Universal Robots URScript: SUB_3100.script

def SUB_3100():
  global _hidden_verificationVariable=0
  set_standard_analog_input_domain(0, 1)
  set_standard_analog_input_domain(1, 1)
  set_tool_analog_input_domain(0, 1)
  set_tool_analog_input_domain(1, 1)
  set_analog_outputdomain(0, 0)
  set_analog_outputdomain(1, 0)
  set_input_actions_to_default()
  set_runstate_gp_boolean_output_to_value(0, 3)
  set_safety_mode_transition_hardness(1)
  set_tcp(p[0.0,0.06,0.535,0.0,0.0,0.0])
  set_gravity([0.0, 0.0, 9.82])
  set_tool_communication(False, 115200, 0, 1, 1.5, 3.5)
  set_tool_output_mode(0)
  set_tool_digital_output_mode(0, 1)
  set_tool_digital_output_mode(1, 1)
  set_tool_voltage(0)
  set_target_payload(0.100000, [0.135000, 0.000000, 0.225000], [10.000000, 10.000000, 10.000000, 0.000000, 0.000000, 0.000000])
  global isReCapt=False
  global Bucket_Z=[0, 0.7]
  global DistPillar=475
  global CandCnt=0
  global lr=1
  global ReCaptZ=0.05
  global forceval=p[0, 0, 0, 0, 0, 0]
  global CaptDepth=[0.24, 0.72, 0]
  global port=3000
  global isOnlyF=True
  global retX2=p[-0.09927, 0.42868, -0.30877, 0.00019, -0.00018, -1.59231]
  global socket_timeout=120
  global isSkipP=False
  global curpos=p[0, 0, 0, 0, 0, 0]
  global host="192.168.1.2"
  global is_popup=False
  global CaptZOffset=0
  global isGoHome=True
  global i_pos2=p[-0.73669, 0.09787, -0.42767, 2.01816, 2.03864, 0.34287]
  global i_pos1=p[-0.73588, 0.09792, -0.42776, 2.01775, 2.03812, 0.34393]
  global pBucket=[p[0.82431, 0.40374, 0.29254, 0, 0, -1.56059], p[-0.84041, -0.48526, 0.27877, 0, 0, 1.6028], p[0, 0, 0, 0, 0, 0]]
  global CaptStepZ=0.08
  global CaptIndex=[0, 0, 0]
  global CaptStepX=0.432
  global pBucketM=p[-0.80141, -0.42542, 0.2879, 0, 0, 1.55713]
  global socket_name="vt"
  global rovi_err=0
  global SubPrgResult=820
  global CurrPos=p[-0.89356, -0.02064, 0.55405, 2.21465, 2.1843, 0.05997]
  global CurrPos_p=p[-0.80753, -0.01858, 0.02262, 2.21465, 2.1843, 0.05997]
  global ForceStartZ=0.43553
  global CutOffZ=0.08
  global HomeDistTh=0.05
  global RBDistTh=0.05
  global RBRadiusTh=0.3
  global RBXTh=[-0.5, 0.5]
  global RBYTh=[-0.8, 1]
  global RBZTh=[-0.1, 0.1]
  global Sub3100_ZMax=0.74
  global ForceStartX=-0.98868
  global Sub3100_aRot=0.2
  global Sub3100_d=0.3
  global Sub3100_Option=18
  global Sub3100_a=0.2
  global Sub3100_XdV=0.1
  global Sub3100_XdRot=8
  global ZoneDistTh=0.05
  global ZoneRadiusTh=0.3
  global ZoneXTh=[-0.5, 0.5]
  global ZoneYTh=[-0.8, 1]
  global ZoneZTh=[-0.1, 0.1]
  global BucketWidth=0.95
  global ZoneBucketGap=0.1
  global ZoneHomeX=[-0.2, 0.2]
  global UnloadZ=0.05
  global CaptPos=p[-0.42193,-0.00317,0.36000,2.199,2.246,0.022]
  global BucketUpperPos=p[0.42193,0.00317,0.36000,2.199,2.246,0.022]
  global Sub3100_GPII18=0
  global Bucket=p[0.32604,0.49174,0.0,-1.882900624652718E-5,2.8304179127934987E-5,-1.593185305749222]
  global BucketM=p[0.32604,0.49174,0.0,1.2814539732933814E-16,-2.611297964559462E-16,-1.5931853071795858]
  global CaptPoint_C=p[-0.4219337985373468,-0.003168602281063755,0.36,-2.1962364319979395,-2.2439316084554193,-0.02184884826814999]
  global CaptPoint_C2=p[0.32796661698047924,-0.010768520544682924,0.01931625281283378,2.2288103429550152,-2.213636886217198,8.598462540813273E-5]
  global CaptPoint_L1=p[-0.42193494849366175,-0.2,0.36,-2.1962086037526616,-2.243896582262281,-0.02199725151102503]
  global CaptPoint_L2=p[0.327894307417917,-0.010799940826224014,0.01928712668893995,2.087717047309385,-2.0736781215133306,0.27365839887453103]
  global CaptPoint_R1=p[-0.4219551896101372,0.3,0.36,-2.1960823751566156,-2.243954123514977,-0.021863042557794844]
  global CaptPoint_R2=p[0.327926308680866,-0.010795166414457658,0.019300245403843563,-2.1186306375223185,2.1040550557443427,0.22023197678473694]
  global Capt_1BK_L=p[-0.4574214308482636,-0.48457071473611046,0.3504487959434708,-2.1962343446504526,-2.243967222238911,-0.021809195357489434]
  global Capt_1BK_L_kari=p[-0.9062780457975316,-0.3948152887685301,0.3041579389647211,-1.973454285761923,-1.9354309814821136,0.46582663599327684]
  global Capt_1BK_R=p[-0.4574597285646511,0.4755214243904677,0.35039311859649847,-2.196330286580149,-2.2438949166739053,-0.021738621025254933]
  global Capt_1BK_R_kari=p[-0.9062432457725078,0.5951337546911526,0.30410336812750105,-1.9735777661712788,-1.9353884348839347,0.46584435471052615]
  global Capt_1BK_pos1=p[-0.4218793038724447,-0.003154429464978058,0.2915499891144615,-2.1963422029204875,-2.2438663520270015,-0.02197160668673838]
  global Capt_1BK_pos2=p[-0.42187829024618434,-0.0031710253373066375,0.29156503858953065,-2.196324918349679,-2.2439040699490773,-0.021928444416953782]
  global Capt_1BK_pos2_k=p[-0.6125678682784722,-0.030388805985305904,0.07817890571333086,-1.7892541925095446,-1.8765982468297469,0.6168577595976025]
  global Capt_2BK_L=p[0.42186661528427194,0.4254738068040517,0.35042275762909847,2.239156309475874,-2.1837044610999294,0.002643817066643282]
  global Capt_2BK_L_kari=p[1.0654977997166857,0.48819520122022786,0.0997150581225536,-1.8581624430714432,1.7479280549699192,-0.330138866280949]
  global Capt_2BK_R=p[0.4218208572756906,-0.5427676723257963,0.350372239919558,2.2392697861179327,-2.183553596194912,0.002410470905346486]
  global Capt_2BK_R_kari=p[1.0635189639466671,-0.5406292885234477,0.09156512141204048,-2.1417082668537115,1.7859902718169367,-0.7309097134650204]
  global Capt_2BK_pos1=p[0.42193501458435656,0.004742683868356356,0.35045865974037793,2.2391012408536453,-2.1839704655717003,0.002677867056024068]
  global Capt_2BK_pos2=p[0.421903984494575,0.004707988774967922,0.35045218900915065,2.239114367170047,-2.183895515396197,0.002684056681074047]
  global Capt_2BK_pos2_k=p[0.4977433025854323,-0.009744988529796803,0.07805101846052531,-1.951106747250682,1.9044153054141988,-0.5362260997480872]
  global Capt_GD_M=p[-0.004067001529315755,-0.25244814937804905,-2.093072695775744E-4,0.0332905748643788,-3.1401478399413327,-0.0037841799742876323]
  global Depart_1GD=p[2.9272629556870893E-4,-0.32809839693864495,0.01933497371622539,0.06378642771012696,-3.140731101950783,-3.370184732371461E-4]
  global Depart_LM_2GD=p[-0.022329487227551487,-0.6428077701737687,0.030336146545121845,-0.0656618547018821,2.9888986438241005,0.1566836156643787]
  global Depart_M=p[0.03703236558231149,-0.6428132409158767,-0.02112384231382136,-0.05669816428100925,3.1320592135794345,0.16829522075932857]
  global Depart_RM_2GD=p[0.10304778501057178,-0.6389514408512296,0.030085893950939302,0.039485966396909634,-3.0126453050861945,-0.17126767917269797]
  global Depsrt_2GD=p[3.027477292580124E-4,-0.3281073069657892,0.019292078494201337,0.06380062875024692,-3.1406974312388685,-3.876005598966342E-4]
  global HomePointL=p[-0.36789,-0.5117344641471838,0.78,-0.6278857271586024,3.0680899128661667,-8.649957362498864E-4]
  global PickPos=p[0.10830682331105715,-1.3709505888096256,-0.18404188875951455,-0.00622194000158997,2.880236948927292,-0.00383636509397631]
  global Solve=p[-0.00368,-0.0021000000000000003,0.25739999999999996,0.0,0.0,0.0]
  global TEST=p[0.1,0.0,0.2,0.0,0.0,0.0]
  global UF=p[0.0,0.0,0.0,0.0,0.0,0.0]
  global g1CV_1_M=p[0.29093319989156785,-0.9405344885124904,-0.08686754932079166,1.9884186265311852,2.2323374792844253,0.1524643645929425]
  global g1CV_posL1=p[0.05028133628211688,-0.4526481033729615,0.1221845548632916,-2.213335080948508,-2.1937561336067057,-0.3280056759040735]
  global g1CV_posR1=p[0.03743870476062511,-0.53119407812668,0.11301901343688614,2.073418671558482,2.153257467049566,0.11656306439039889]
  global g1GD_pos1=p[0.06841781024889843,-0.5456037307108855,0.367146167315866,2.4108578981103275,1.7957834606331096,0.12544942012730473]
  global g1GD_pos2=p[-0.38705506163240566,-0.3905161646272917,0.3670805000411974,2.9334800678601534,0.5562338866571123,0.025147235284150155]
  global g1GD_pos3=p[-0.614523200343285,-0.009392732880809615,0.3783325239377683,2.0687271625579515,2.17319336139756,0.21682066343437634]
  global g1GD_pos4=p[-0.4351564513137486,0.028155221259926276,0.13086718327275837,2.2072871432536783,2.2307343865376095,-0.0018307218179379997]
  global g1GD_pos5=p[-0.8151645021025727,-0.01706756320728201,0.08179601375099321,2.212895896456039,2.218350348620789,0.019350113017735118]
  global g1GD_posL1=p[-0.08276848269606216,-0.3996147100031649,0.1488453551331823,2.286527078917204,1.8420745504477611,0.33698451773695576]
  global g1GD_posL2=p[-0.3253977027403738,-0.3024804624281039,0.16332814085945146,2.72312820760317,0.9631021078169197,0.32447452035226126]
  global g1GD_posL3=p[-0.6791033397183219,0.06787475590683856,0.16337212788108813,2.1383125299263996,2.086116032377724,0.4536080263755059]
  global g1GD_posR1=p[-0.09893370538053747,-0.4999608954567234,0.14329885217724153,2.43311852414254,1.4238397520832589,0.08559216753941556]
  global g1GD_posR2=p[-0.3729565201882258,-0.3752983669473301,0.143299052800563,2.6951655216297596,0.8130506811102118,-0.02387549506099888]
  global g1GD_posR3=p[-0.7385929502572233,-0.029472684480355026,0.1499650660949685,2.0484522752014467,1.9493695704119496,0.18368227556562683]
  global g2CV_1_M=p[0.2880593256931911,-0.933809998732841,-0.08698643380656113,2.0727630257838867,2.230596497566155,0.15036691287620893]
  global g2CV_posL1=p[0.3409386496330911,-0.4656338066361442,0.1250074988128972,2.209372209162659,2.1945371304665926,0.3160714960040194]
  global g2CV_posR1=p[0.3400736278759575,-0.531334269888987,0.1183415684753657,2.07314649492589,2.1532617466521136,0.11638666128062146]
  global g2GD_pos1=p[0.3390086633742754,-0.5203839341398588,0.22258,2.022696172282159,2.259224887850344,0.09811005079237367]
  global g2GD_pos2=p[0.4140891885236144,0.14850105084950693,0.1582916370575993,-0.10302503203970696,3.1008909166713883,0.18748967846962497]
  global g2GD_pos3=p[0.32377086541216454,-0.01023215987367155,0.15821240334102793,2.279746475463588,-2.06129961332614,-0.16578334012307952]
  global g2GD_pos4=p[0.7398823109797592,-0.026643494293930835,0.22255839224074236,2.162283599874437,-2.168919538925757,-0.13861635932587069]
  global g2GD_pos5=p[0.22271243238356278,-0.026679271241024524,0.22257782526136982,1.3056143664331146,-2.8077458860488136,-0.17177240522535248]
  global gCV_11_M=p[0.3028468774759881,-0.9375366886748661,-0.09782511939875749,1.9971971468330036,2.0934336167121885,0.3604928446251781]
  global gCV_12_M=p[0.34776610649632045,-0.9364202289953052,-0.09784932758070936,1.9972781240484352,2.0934384510830295,0.3604701319279358]
  global gCV_13_M=p[0.43083047728791135,-0.9363258116427577,0.028711300566433673,1.9972504931093251,2.0935710325846095,0.3605630596092243]
  global gCV_14=p[0.35645641620611146,-0.8914305774826713,-0.17737239800677018,2.1506886654737776,2.1461343800624295,0.40986447399780934]
  global gCV_15=p[0.4370373250739419,-0.891408661166693,-0.1773997714481486,2.1507483614991094,2.1461657601704176,0.40983132876462236]
  global gCV_16=p[0.4597123429384979,-0.8913837618729653,-0.03599504377258328,2.1506156333226136,2.1462305295546718,0.4099109158136618]
  global gCV_17=p[0.037528034463104695,-0.6904892259828748,-0.12243237639232962,-0.12012393052395552,2.832430475095037,0.48967048060305135]
  global gCV_18=p[0.03600103065313248,-0.6368623043127666,-0.12241687036449483,-0.12010351348807546,2.832474314609516,0.48970816626953567]
  global gCV_2_M=p[0.2909259851094176,-0.9405632657218349,0.07217586581493451,1.9883998690824036,2.232303337331875,0.15240099649164607]
  global gCV_3_M=p[0.29099390607376485,-0.6570558385379063,0.0722153583041818,1.9884242634571576,2.2321538498123994,0.15249643504377583]
  global gCV_5=p[0.045776199142861046,-0.9791473230816141,0.8415069045351792,2.0229894037377316,2.080009888728606,0.35618099403901887]
  global gCV_pos5=p[0.3400172856834047,-0.9722754606605235,-0.18287928563575456,2.073394561413637,2.1531827558666565,0.11639000988241816]
  global gGD_100_1LM=p[0.04146780808756359,-0.6870904124925177,-0.1232943093634104,-0.006305250057386166,-2.863965809273829,-0.5082528300185785]
  global gGD_1_LM=p[0.03230475520524248,-0.7130493639313011,-0.12313048496237139,-0.146861070648958,2.82789794799972,0.5264874367071143]
  global gGD_1_M=p[0.03530347986661216,-0.7127417041043018,-0.12310155616185803,-0.05957601747684272,3.087266550524023,0.5413331493142363]
  global gGD_1_MM=p[0.03527332731929103,-0.7200324399236822,-0.12309145975746483,-0.05946537723025455,3.087281488106925,0.5412792107775745]
  global gGD_1_RM=p[0.03790072787181614,-0.7120178370098972,-0.12342664631367783,0.016248473772828512,-2.8629005997783534,-0.4984191911686871]
  global gGD_200_2LM=p[0.04175812558137225,-0.6358261219893102,-0.12285474020423298,-0.006257718193554584,-2.863964784148567,-0.5084621939645108]
  global gGD_2_LM=p[0.030572718129261614,-0.6604571464977577,-0.12310155388330796,-0.14682775034190318,2.827796436074414,0.5264394416290918]
  global gGD_2_M=p[0.03435287261256309,-0.6587000226205477,-0.12439339172019714,-0.05966040009453588,3.0872872080206544,0.5411228747416044]
  global gGD_2_RM=p[0.036719806244467246,-0.6603323308238997,-0.12407566124392316,0.01621270878011713,-2.862858880050919,-0.4984088290677938]
  global gGD_300_3LM=p[0.04182050265947469,-0.6066076810742604,-0.03602288107395374,-0.006290924000441408,-2.8640915241774816,-0.5083501301248439]
  global gGD_3_LM=p[0.03053842874056699,-0.6329626532416066,-0.03639755844951337,-0.14684511442606807,2.8278657439893307,0.5264948582193963]
  global gGD_3_M=p[0.03430957843779042,-0.6330568980917707,-0.04259950182125549,-0.05969688861307265,3.087293602983763,0.5413247841490268]
  global gGD_3_RM=p[0.03673432946585267,-0.632032638942058,-0.03445023119106272,0.016317873028914045,-2.8628788700289953,-0.4985371510851901]
  global gGD_400_1RM=p[0.03765496539143813,-0.6905733748742057,-0.12240702670509729,-0.12009639012349203,2.8324503628258273,0.48945657912051843]
  global gGD_4_LM=p[-0.050697518013391604,-0.4788149830819543,0.04525080740157289,-0.14673385744666134,2.827848291285266,0.5267055795817903]
  global gGD_4_RM=p[0.10921584432919978,-0.48073334437858256,0.06990685637741062,0.016338390530391603,-2.862804566994448,-0.49861203356258266]
  global gGD_500_2RM=p[0.0364038044475721,-0.6361408639594927,-0.1228896102948493,-0.12001814478849077,2.8324363686538967,0.4895422385690364]
  global gGD_600_3RM=p[0.03597788557419286,-0.6039591135870097,-0.03251312847845622,-0.12016380804709932,2.832584395249392,0.4895204315491753]
  global gGD_M_20=p[0.03524102305764369,-0.704963855446233,-0.12310321086399345,-0.05961230604660993,3.0873078767639504,0.5414261100507907]
  global gGD_M_30=p[0.03527181411394771,-0.6949613298581867,-0.12309199448652725,-0.05962447301074729,3.087287038166274,0.5412100180254447]
  global gGD_M_40=p[0.035236425258241534,-0.6834410208824955,-0.12309554834290798,-0.05953064339288712,3.087315110349415,0.5412921265180426]
  global gHome_Position=p[3.053061697190075E-4,-0.3281132156787397,0.01930332806480972,0.0637196994340987,-3.140722020313799,-3.2847660283345163E-4]
  # begin: URCap Installation Node
  #   Source: Ethernet/IP I/O Monitor URCap, 1.0.0,
  #   Type: Ethernet/IP I/O Monitor
  conn = rpc_factory("xmlrpc", "http://127.0.0.1:" + to_str(61101) + "/RPC2")

  def show_monitor():
    return conn.eip_monitor.show()
  end
  # end: URCap Installation Node
  step_count_5b8865bc_2e57_47ac_841d_e2d67d0170a2 = 0.0
  thread Step_Counter_Thread_a1e906e4_ec48_4bf5_b1d6_2891aa203b67():
    while (True):
      step_count_5b8865bc_2e57_47ac_841d_e2d67d0170a2 = step_count_5b8865bc_2e57_47ac_841d_e2d67d0170a2 + 1.0
      sync()
    end
  end
  run Step_Counter_Thread_a1e906e4_ec48_4bf5_b1d6_2891aa203b67()
  while (True):
    $ 2 "ロボットプログラム"
    $ 3 "ループ"
    while (True):
      $ 4 "Sub3100_Option:=Sub3100_GPII18"
      global Sub3100_Option=Sub3100_GPII18
      $ 5 "If文 (Sub3100_Option≤14)"
      if ((Sub3100_Option <= 14)):
        $ 6 "'MOVE'"
        # 'MOVE'
        $ 7 "If文 GPBI_PrgRun"
        global thread_flag_7=0
        thread Thread_if_7():
          $ 8 "設定 GPBO_PrgRun= True "
          write_output_boolean_register(6,   True  )
          $ 9 "If文 GPBI_BLLoad1"
          if (read_input_boolean_register(10)):
            $ 10 "If文 (1≤Sub3100_Option and Sub3100_Option≤4)"
            if ((1 <= Sub3100_Option  and  Sub3100_Option <= 4)):
              $ 11 "荷重の設定: k10"
              set_target_payload(0.100000, [0.135000, 0.000000, 0.225000], [10.000000, 10.000000, 10.000000, 0.000000, 0.000000, 0.000000])
            else:
              $ 12 "ElseIf (5≤Sub3100_Option and Sub3100_Option≤6)"
              if ((5 <= Sub3100_Option  and  Sub3100_Option <= 6)):
                $ 13 "荷重の設定: k120"
                set_target_payload(0.100000, [0.135000, 0.000000, 0.225000], [120.000000, 120.000000, 120.000000, 0.000000, 0.000000, 0.000000])
              else:
                $ 14 "ElseIf (7≤Sub3100_Option and Sub3100_Option≤12)"
                if ((7 <= Sub3100_Option  and  Sub3100_Option <= 12)):
                  $ 15 "荷重の設定: k10"
                  set_target_payload(0.100000, [0.135000, 0.000000, 0.225000], [10.000000, 10.000000, 10.000000, 0.000000, 0.000000, 0.000000])
                else:
                  $ 16 "ElseIf (13≤Sub3100_Option and Sub3100_Option≤14)"
                  if ((13 <= Sub3100_Option  and  Sub3100_Option <= 14)):
                    $ 17 "荷重の設定: k10"
                    set_target_payload(0.100000, [0.135000, 0.000000, 0.225000], [10.000000, 10.000000, 10.000000, 0.000000, 0.000000, 0.000000])
                  end
                end
              end
            end
          else:
            $ 18 "Else" "noBreak"
            $ 19 "If文 (1≤Sub3100_Option and Sub3100_Option≤4)"
            if ((1 <= Sub3100_Option  and  Sub3100_Option <= 4)):
              $ 20 "荷重の設定: k10"
              set_target_payload(0.100000, [0.135000, 0.000000, 0.225000], [10.000000, 10.000000, 10.000000, 0.000000, 0.000000, 0.000000])
            else:
              $ 21 "ElseIf (5≤Sub3100_Option and Sub3100_Option≤6)"
              if ((5 <= Sub3100_Option  and  Sub3100_Option <= 6)):
                $ 22 "荷重の設定: k120"
                set_target_payload(0.100000, [0.135000, 0.000000, 0.225000], [120.000000, 120.000000, 120.000000, 0.000000, 0.000000, 0.000000])
              else:
                $ 23 "ElseIf (7≤Sub3100_Option and Sub3100_Option≤12)"
                if ((7 <= Sub3100_Option  and  Sub3100_Option <= 12)):
                  $ 24 "荷重の設定: k10"
                  set_target_payload(0.100000, [0.135000, 0.000000, 0.225000], [10.000000, 10.000000, 10.000000, 0.000000, 0.000000, 0.000000])
                else:
                  $ 25 "ElseIf (13≤Sub3100_Option and Sub3100_Option≤14)"
                  if ((13 <= Sub3100_Option  and  Sub3100_Option <= 14)):
                    $ 26 "荷重の設定: k10"
                    set_target_payload(0.100000, [0.135000, 0.000000, 0.225000], [10.000000, 10.000000, 10.000000, 0.000000, 0.000000, 0.000000])
                  end
                end
              end
            end
          end
          $ 27 "ループ"
          while (True):
            $ 28 "Sub3100_Xd:=[0.,0.,0.,0.,0.,0.]"
            global Sub3100_Xd=[0.,0.,0.,0.,0.,0.]
            $ 29 "Sub3100_q:=floor((Sub3100_Option-1) / 2)"
            global Sub3100_q=floor((Sub3100_Option-1) / 2)
            $ 30 "Sub3100_e:=1-((Sub3100_Option-1) % 2)*2"
            global Sub3100_e=1-((Sub3100_Option-1) % 2)*2
            $ 31 "Sub3100_t:=0.5"
            global Sub3100_t=0.5
            $ 32 "If文 (1≤Sub3100_Option and Sub3100_Option≤6)"
            if ((1 <= Sub3100_Option  and  Sub3100_Option <= 6)):
              $ 33 "'1:X+,2:X-,3:Y+,4:Y-,5:Z+,6:Z-'"
              # '1:X+,2:X-,3:Y+,4:Y-,5:Z+,6:Z-'
              $ 34 "Sub3100_Xd[Sub3100_q]=Sub3100_XdV*Sub3100_e"
              Sub3100_Xd[Sub3100_q]=Sub3100_XdV*Sub3100_e
              $ 35 "If文 Sub3100_Option≟5"
              if (Sub3100_Option == 5):
                $ 36 "If文 CurrPos[2]<Sub3100_ZMax"
                global thread_flag_36=0
                thread Thread_if_36():
                  $ 37 "speedl(Sub3100_Xd,Sub3100_a,t=Sub3100_t)"
                  speedl(Sub3100_Xd,Sub3100_a,t=Sub3100_t)
                  thread_flag_36 = 1
                end
                if (CurrPos[2]<Sub3100_ZMax):
                  global thread_handler_36=run Thread_if_36()
                  while (thread_flag_36 == 0):
                    if not(CurrPos[2]<Sub3100_ZMax):
                      kill thread_handler_36
                      thread_flag_36 = 2
                    else:
                      sync()
                    end
                  end
                else:
                  thread_flag_36 = 2
                end
                $ 38 "stopl(Sub3100_d)"
                stopl(Sub3100_d)
              else:
                $ 39 "Else" "noBreak"
                $ 40 "speedl(Sub3100_Xd,Sub3100_a,t=Sub3100_t)"
                speedl(Sub3100_Xd,Sub3100_a,t=Sub3100_t)
              end
            else:
              $ 41 "ElseIf (7≤Sub3100_Option and Sub3100_Option≤12)"
              if ((7 <= Sub3100_Option  and  Sub3100_Option <= 12)):
                $ 42 "'7:RX+,8:RX-,9:RY+,10:RY-,11:RZ+,12:RZ-'"
                # '7:RX+,8:RX-,9:RY+,10:RY-,11:RZ+,12:RZ-'
                $ 43 "Sub3100_Xd[Sub3100_q]=d2r(Sub3100_XdRot)*Sub3100_e"
                Sub3100_Xd[Sub3100_q]= d2r (Sub3100_XdRot)*Sub3100_e
                $ 44 "speedl(Sub3100_Xd,Sub3100_aRot,Sub3100_t)"
                speedl(Sub3100_Xd,Sub3100_aRot,Sub3100_t)
              else:
                $ 45 "ElseIf (Sub3100_Option≟13 or Sub3100_Option≟14)"
                if ((Sub3100_Option == 13  or  Sub3100_Option == 14)):
                  $ 46 "'13:TZ+,14:TZ-'"
                  # '13:TZ+,14:TZ-'
                  $ 47 "Sub3100_curr:=CurrPos_p"
                  global Sub3100_curr=CurrPos_p
                  $ 48 "var_1:=p[0.,0.,0.,0.,0.,0.]"
                  global var_1=p[0.,0.,0.,0.,0.,0.]
                  $ 49 "var_1[Sub3100_q-4]=0.25*Sub3100_e"
                  var_1[Sub3100_q-4]=0.25*Sub3100_e
                  $ 50 "var_2:=pose_sub(pose_trans(Sub3100_curr,var_1),Sub3100_curr)"
                  global var_2= pose_sub (pose_trans(Sub3100_curr,var_1),Sub3100_curr)
                  $ 51 "ループ6回"
                  u12523u12540u12503_3 = 0
                  while (u12523u12540u12503_3 < 6):
                    $ 52 "Sub3100_Xd[ループ_8]=var_2[ループ_8]"
                    Sub3100_Xd[u12523u12540u12503_8]=var_2[u12523u12540u12503_8]
                    u12523u12540u12503_3 = u12523u12540u12503_3 + 1
                  end
                  $ 53 "speedl(Sub3100_Xd,Sub3100_a,Sub3100_t)"
                  speedl(Sub3100_Xd,Sub3100_a,Sub3100_t)
                end
              end
            end
          end
          thread_flag_7 = 1
        end
        if (read_input_boolean_register(6)):
          global thread_handler_7=run Thread_if_7()
          while (thread_flag_7 == 0):
            if not(read_input_boolean_register(6)):
              kill thread_handler_7
              thread_flag_7 = 2
            else:
              sync()
            end
          end
        else:
          thread_flag_7 = 2
        end
        $ 54 "stopl(Sub3100_d)"
        stopl(Sub3100_d)
      else:
        $ 55 "ElseIf (Sub3100_Option≤44)"
        if ((Sub3100_Option <= 44)):
          $ 56 "'FORCE'"
          # 'FORCE'
          $ 57 "If文 GPBI_PrgRun"
          if (read_input_boolean_register(6)):
            $ 58 "設定 GPBO_PrgRun= True "
            write_output_boolean_register(6,   True  )
            $ 59 "If文 GPBI_BLLoad1"
            if (read_input_boolean_register(10)):
              $ 60 "If文 (33≤Sub3100_Option and Sub3100_Option≤36)"
              if ((33 <= Sub3100_Option  and  Sub3100_Option <= 36)):
                $ 61 "荷重の設定: k05"
                set_target_payload(0.100000, [0.135000, 0.000000, 0.255000], [0.500000, 0.500000, 0.500000, 0.000000, 0.000000, 0.000000])
              else:
                $ 62 "ElseIf (37≤Sub3100_Option and Sub3100_Option≤38)"
                if ((37 <= Sub3100_Option  and  Sub3100_Option <= 38)):
                  $ 63 "荷重の設定: k05"
                  set_target_payload(0.100000, [0.135000, 0.000000, 0.255000], [0.500000, 0.500000, 0.500000, 0.000000, 0.000000, 0.000000])
                else:
                  $ 64 "ElseIf (39≤Sub3100_Option and Sub3100_Option≤44)"
                  if ((39 <= Sub3100_Option  and  Sub3100_Option <= 44)):
                    $ 65 "荷重の設定: k05"
                    set_target_payload(0.100000, [0.135000, 0.000000, 0.255000], [0.500000, 0.500000, 0.500000, 0.000000, 0.000000, 0.000000])
                  end
                end
              end
            else:
              $ 66 "Else" "noBreak"
              $ 67 "If文 (33≤Sub3100_Option and Sub3100_Option≤36)"
              if ((33 <= Sub3100_Option  and  Sub3100_Option <= 36)):
                $ 68 "荷重の設定: k05"
                set_target_payload(0.100000, [0.135000, 0.000000, 0.255000], [0.500000, 0.500000, 0.500000, 0.000000, 0.000000, 0.000000])
              else:
                $ 69 "ElseIf (37≤Sub3100_Option and Sub3100_Option≤38)"
                if ((37 <= Sub3100_Option  and  Sub3100_Option <= 38)):
                  $ 70 "荷重の設定: k05"
                  set_target_payload(0.100000, [0.135000, 0.000000, 0.255000], [0.500000, 0.500000, 0.500000, 0.000000, 0.000000, 0.000000])
                else:
                  $ 71 "ElseIf (39≤Sub3100_Option and Sub3100_Option≤44)"
                  if ((39 <= Sub3100_Option  and  Sub3100_Option <= 44)):
                    $ 72 "荷重の設定: k05"
                    set_target_payload(0.100000, [0.135000, 0.000000, 0.255000], [0.500000, 0.500000, 0.500000, 0.000000, 0.000000, 0.000000])
                  end
                end
              end
            end
            $ 73 "If文 (Sub3100_Option≟33)"
            if ((Sub3100_Option == 33)):
              $ 74 "'33:X+'"
              # '33:X+'
              $ 75 "フォース"
              sleep(0.02)
              zero_ftsensor()
              force_mode(p[0.0,0.0,0.0,0.0,0.0,0.0], [1, 1, 1, 1, 1, 1], [40.0, 0.0, 0.0, 0.0, 0.0, 0.0], 2, [0.01, 0.005, 0.005, 0.03490658503988659, 0.03490658503988659, 0.03490658503988659])
              $ 76 "待機 GPBI_PrgRun=LO" "noBreak"
              while (read_input_boolean_register(6) == True):
                sync()
              end
              end_force_mode()
              stopl(5.0)
            else:
              $ 77 "ElseIf (Sub3100_Option≟34)"
              if ((Sub3100_Option == 34)):
                $ 78 "'34:X-'"
                # '34:X-'
                $ 79 "フォース"
                sleep(0.02)
                zero_ftsensor()
                force_mode(p[0.0,0.0,0.0,0.0,0.0,0.0], [1, 1, 1, 1, 1, 1], [-40.0, 0.0, 0.0, 0.0, 0.0, 0.0], 2, [0.01, 0.005, 0.005, 0.03490658503988659, 0.03490658503988659, 0.03490658503988659])
                $ 80 "待機 GPBI_PrgRun=LO" "noBreak"
                while (read_input_boolean_register(6) == True):
                  sync()
                end
                end_force_mode()
                stopl(5.0)
              else:
                $ 81 "ElseIf (Sub3100_Option≟35)"
                if ((Sub3100_Option == 35)):
                  $ 82 "'35:Y+'"
                  # '35:Y+'
                  $ 83 "フォース"
                  sleep(0.02)
                  zero_ftsensor()
                  force_mode(p[0.0,0.0,0.0,0.0,0.0,0.0], [1, 1, 1, 1, 1, 1], [0.0, 40.0, 0.0, 0.0, 0.0, 0.0], 2, [0.005, 0.01, 0.005, 0.03490658503988659, 0.03490658503988659, 0.03490658503988659])
                  $ 84 "待機 GPBI_PrgRun=LO" "noBreak"
                  while (read_input_boolean_register(6) == True):
                    sync()
                  end
                  end_force_mode()
                  stopl(5.0)
                else:
                  $ 85 "ElseIf (Sub3100_Option≟36)"
                  if ((Sub3100_Option == 36)):
                    $ 86 "'36:Y-'"
                    # '36:Y-'
                    $ 87 "フォース"
                    sleep(0.02)
                    zero_ftsensor()
                    force_mode(p[0.0,0.0,0.0,0.0,0.0,0.0], [1, 1, 1, 1, 1, 1], [0.0, -40.0, 0.0, 0.0, 0.0, 0.0], 2, [0.005, 0.01, 0.005, 0.03490658503988659, 0.03490658503988659, 0.03490658503988659])
                    $ 88 "待機 GPBI_PrgRun=LO" "noBreak"
                    while (read_input_boolean_register(6) == True):
                      sync()
                    end
                    end_force_mode()
                    stopl(5.0)
                  else:
                    $ 89 "ElseIf (Sub3100_Option≟37)"
                    if ((Sub3100_Option == 37)):
                      $ 90 "'37:Z+'"
                      # '37:Z+'
                      $ 91 "フォース"
                      sleep(0.02)
                      zero_ftsensor()
                      force_mode(p[0.0,0.0,0.0,0.0,0.0,0.0], [1, 1, 1, 1, 1, 1], [0.0, 0.0, 40.0, 0.0, 0.0, 0.0], 2, [0.005, 0.005, 0.01, 0.03490658503988659, 0.03490658503988659, 0.03490658503988659])
                      $ 92 "待機 GPBI_PrgRun=LO" "noBreak"
                      while (read_input_boolean_register(6) == True):
                        sync()
                      end
                      end_force_mode()
                      stopl(5.0)
                    else:
                      $ 93 "ElseIf (Sub3100_Option≟38)"
                      if ((Sub3100_Option == 38)):
                        $ 94 "'38:Z-'"
                        # '38:Z-'
                        $ 95 "フォース"
                        sleep(0.02)
                        zero_ftsensor()
                        force_mode(p[0.0,0.0,0.0,0.0,0.0,0.0], [1, 1, 1, 1, 1, 1], [0.0, 0.0, -40.0, 0.0, 0.0, 0.0], 2, [0.005, 0.005, 0.01, 0.03490658503988659, 0.03490658503988659, 0.03490658503988659])
                        $ 96 "待機 GPBI_PrgRun=LO" "noBreak"
                        while (read_input_boolean_register(6) == True):
                          sync()
                        end
                        end_force_mode()
                        stopl(5.0)
                      else:
                        $ 97 "ElseIf (Sub3100_Option≟39)"
                        if ((Sub3100_Option == 39)):
                          $ 98 "'39:RX+'"
                          # '39:RX+'
                          $ 99 "フォース"
                          sleep(0.02)
                          zero_ftsensor()
                          force_mode(p[0.0,0.0,0.0,0.0,0.0,0.0], [1, 1, 1, 1, 1, 1], [0.0, 0.0, 0.0, 40.0, 0.0, 0.0], 2, [0.005, 0.005, 0.005, 0.08726646259971647, 0.03490658503988659, 0.03490658503988659])
                          $ 100 "待機 GPBI_PrgRun=LO" "noBreak"
                          while (read_input_boolean_register(6) == True):
                            sync()
                          end
                          end_force_mode()
                          stopl(5.0)
                        else:
                          $ 101 "ElseIf (Sub3100_Option≟40)"
                          if ((Sub3100_Option == 40)):
                            $ 102 "'40:RX-'"
                            # '40:RX-'
                            $ 103 "フォース"
                            sleep(0.02)
                            zero_ftsensor()
                            force_mode(p[0.0,0.0,0.0,0.0,0.0,0.0], [1, 1, 1, 1, 1, 1], [0.0, 0.0, 0.0, -40.0, 0.0, 0.0], 2, [0.005, 0.005, 0.005, 0.08726646259971647, 0.03490658503988659, 0.03490658503988659])
                            $ 104 "待機 GPBI_PrgRun=LO" "noBreak"
                            while (read_input_boolean_register(6) == True):
                              sync()
                            end
                            end_force_mode()
                            stopl(5.0)
                          else:
                            $ 105 "ElseIf (Sub3100_Option≟41)"
                            if ((Sub3100_Option == 41)):
                              $ 106 "'41:RY+'"
                              # '41:RY+'
                              $ 107 "フォース"
                              sleep(0.02)
                              zero_ftsensor()
                              force_mode(p[0.0,0.0,0.0,0.0,0.0,0.0], [1, 1, 1, 1, 1, 1], [0.0, 0.0, 0.0, 0.0, 40.0, 0.0], 2, [0.005, 0.005, 0.005, 0.03490658503988659, 0.08726646259971647, 0.03490658503988659])
                              $ 108 "待機 GPBI_PrgRun=LO" "noBreak"
                              while (read_input_boolean_register(6) == True):
                                sync()
                              end
                              end_force_mode()
                              stopl(5.0)
                            else:
                              $ 109 "ElseIf (Sub3100_Option≟42)"
                              if ((Sub3100_Option == 42)):
                                $ 110 "'42:RY-'"
                                # '42:RY-'
                                $ 111 "フォース"
                                sleep(0.02)
                                zero_ftsensor()
                                force_mode(p[0.0,0.0,0.0,0.0,0.0,0.0], [1, 1, 1, 1, 1, 1], [0.0, 0.0, 0.0, 0.0, -40.0, 0.0], 2, [0.005, 0.005, 0.005, 0.03490658503988659, 0.08726646259971647, 0.03490658503988659])
                                $ 112 "待機 GPBI_PrgRun=LO" "noBreak"
                                while (read_input_boolean_register(6) == True):
                                  sync()
                                end
                                end_force_mode()
                                stopl(5.0)
                              else:
                                $ 113 "ElseIf (Sub3100_Option≟43)"
                                if ((Sub3100_Option == 43)):
                                  $ 114 "'43:RZ+'"
                                  # '43:RZ+'
                                  $ 115 "フォース"
                                  sleep(0.02)
                                  zero_ftsensor()
                                  force_mode(p[0.0,0.0,0.0,0.0,0.0,0.0], [1, 1, 1, 1, 1, 1], [0.0, 0.0, 0.0, 0.0, 0.0, 40.0], 2, [0.005, 0.005, 0.005, 0.03490658503988659, 0.03490658503988659, 0.08726646259971647])
                                  $ 116 "待機 GPBI_PrgRun=LO" "noBreak"
                                  while (read_input_boolean_register(6) == True):
                                    sync()
                                  end
                                  end_force_mode()
                                  stopl(5.0)
                                else:
                                  $ 117 "ElseIf (Sub3100_Option≟44)"
                                  if ((Sub3100_Option == 44)):
                                    $ 118 "'44:RZ-'"
                                    # '44:RZ-'
                                    $ 119 "フォース"
                                    sleep(0.02)
                                    zero_ftsensor()
                                    force_mode(p[0.0,0.0,0.0,0.0,0.0,0.0], [1, 1, 1, 1, 1, 1], [0.0, 0.0, 0.0, 0.0, 0.0, -40.0], 2, [0.005, 0.005, 0.005, 0.03490658503988659, 0.03490658503988659, 0.08726646259971647])
                                    $ 120 "待機 GPBI_PrgRun=LO" "noBreak"
                                    while (read_input_boolean_register(6) == True):
                                      sync()
                                    end
                                    end_force_mode()
                                    stopl(5.0)
                                  end
                                end
                              end
                            end
                          end
                        end
                      end
                    end
                  end
                end
              end
            end
          end
        else:
          $ 121 "ElseIf (Sub3100_Option≥90)"
          if ((Sub3100_Option >= 90)):
            $ 122 "'FREEDRIVE'"
            # 'FREEDRIVE'
            $ 123 "If文 GPBI_PrgRun"
            if (read_input_boolean_register(6)):
              $ 124 "設定 GPBO_PrgRun= True "
              write_output_boolean_register(6,   True  )
              $ 125 "If文 GPBI_BLLoad1"
              if (read_input_boolean_register(10)):
                $ 126 "荷重の設定: k05"
                set_target_payload(0.100000, [0.135000, 0.000000, 0.255000], [0.500000, 0.500000, 0.500000, 0.000000, 0.000000, 0.000000])
              else:
                $ 127 "Else" "noBreak"
                $ 128 "荷重の設定: k05"
                set_target_payload(0.100000, [0.135000, 0.000000, 0.255000], [0.500000, 0.500000, 0.500000, 0.000000, 0.000000, 0.000000])
              end
              $ 129 "If文 (Sub3100_Option≟90)"
              if ((Sub3100_Option == 90)):
                $ 130 "'90:FreeDrive'"
                # '90:FreeDrive'
                $ 131 "freedrive_mode()"
                freedrive_mode()
                $ 132 "待機 GPBI_PrgRun=LO"
                while (read_input_boolean_register(6) == True):
                  sync()
                end
                $ 133 "end_freedrive_mode()"
                end_freedrive_mode()
              end
            end
          end
        end
      end
      $ 134 "stopl(Sub3100_d)"
      stopl(Sub3100_d)
      $ 135 "待機: 0.01"
      sleep(0.01)
      $ 136 "荷重の設定: k10"
      set_target_payload(0.100000, [0.135000, 0.000000, 0.225000], [10.000000, 10.000000, 10.000000, 0.000000, 0.000000, 0.000000])
      $ 137 "設定 GPBO_PrgRun= False "
      write_output_boolean_register(6,   False  )
    end
  end
end
